Fanuc KAREL source: kb00187.KL

PROGRAM KB00187
%NOLOCKGROUP
VAR
P1:REAL;RESULT:REAL
BEGIN
--
P1=1.0
RESULT=SQRT(P1)
END KB00187
